FUNCTION_BLOCK FACTORY_IO_PICK_AND_PLACE_ROBOT
  {SET_ATTRIBUTE(OpcUa, SERVICE)}
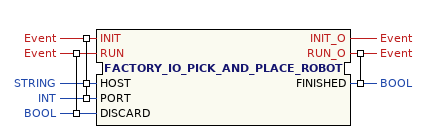
  EVENT_INPUT
    INIT WITH HOST, PORT;
    RUN WITH DISCARD;
  END_EVENT
  EVENT_OUTPUT
    INIT_O;
    RUN_O WITH FINISHED;
  END_EVENT
  VAR_INPUT
    HOST : STRING; {SET_ATTRIBUTE(OpcUa, Constant.RUN)}
    PORT : INT; {SET_ATTRIBUTE(OpcUa, Constant.RUN)}
    DISCARD : BOOL; {SET_ATTRIBUTE(OpcUa, Variable.RUN)}
  END_VAR
  VAR_OUTPUT
    FINISHED : BOOL; {SET_ATTRIBUTE(OpcUa, Variable.RUN)}
  END_VAR
END_FUNCTION_BLOCK
